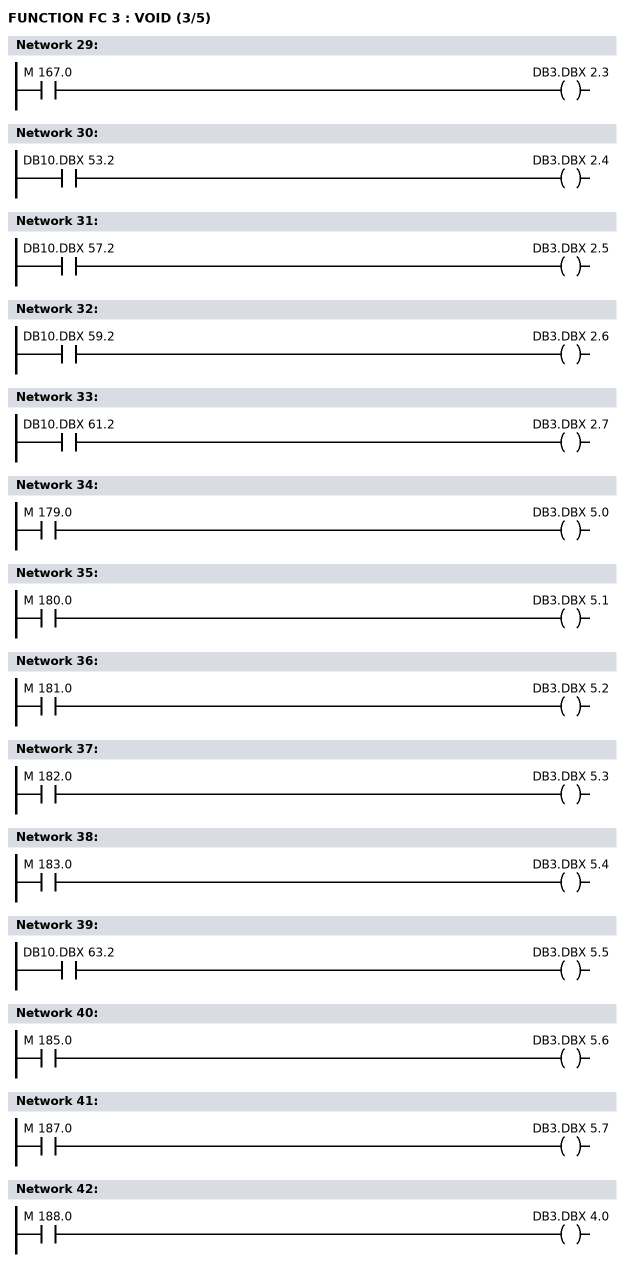

      A     M    167.0;
      =     DB3.DBX    2.3;
NETWORK
TITLE =

      A     DB10.DBX   53.2;
      =     DB3.DBX    2.4;
NETWORK
TITLE =

      A     DB10.DBX   57.2;
      =     DB3.DBX    2.5;
NETWORK
TITLE =

      A     DB10.DBX   59.2;
      =     DB3.DBX    2.6;
NETWORK
TITLE =

      A     DB10.DBX   61.2;
      =     DB3.DBX    2.7;
NETWORK
TITLE =

      A     M    179.0;
      =     DB3.DBX    5.0;
NETWORK
TITLE =

      A     M    180.0;
      =     DB3.DBX    5.1;
NETWORK
TITLE =

      A     M    181.0;
      =     DB3.DBX    5.2;
NETWORK
TITLE =

      A     M    182.0;
      =     DB3.DBX    5.3;
NETWORK
TITLE =

      A     M    183.0;
      =     DB3.DBX    5.4;
NETWORK
TITLE =

      A     DB10.DBX   63.2;
      =     DB3.DBX    5.5;
NETWORK
TITLE =

      A     M    185.0;
      =     DB3.DBX    5.6;
NETWORK
TITLE =

      A     M    187.0;
      =     DB3.DBX    5.7;
NETWORK
TITLE =

      A     M    188.0;
      =     DB3.DBX    4.0;
NETWORK
TITLE =
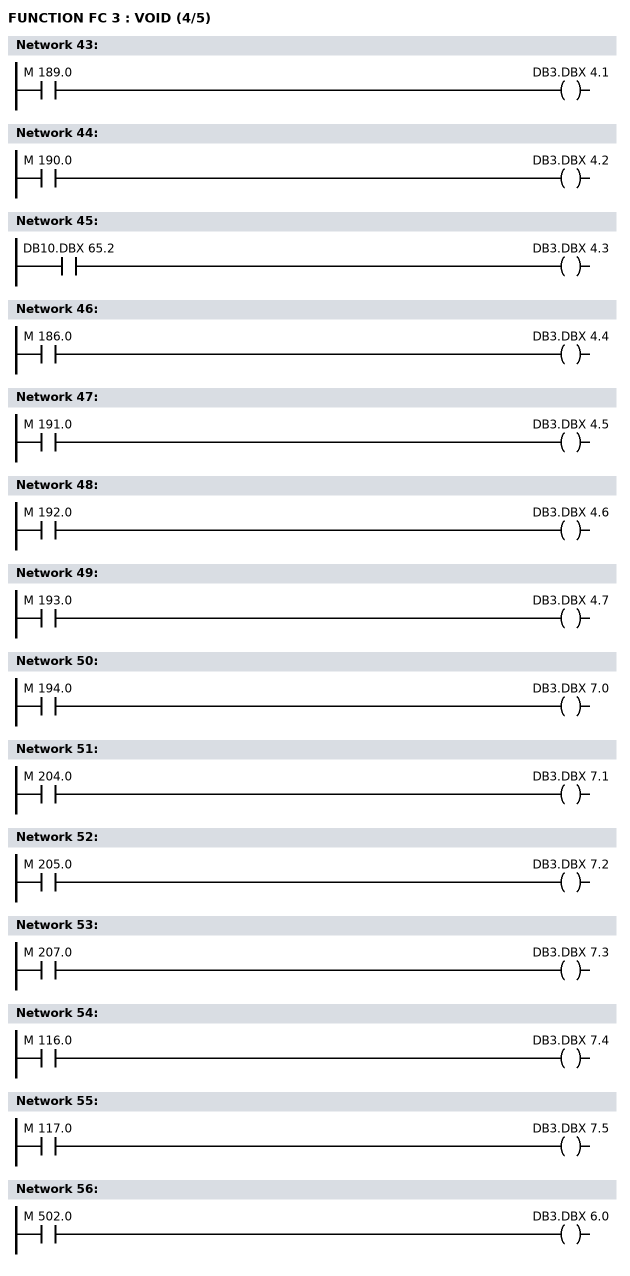

      A     M    189.0;
      =     DB3.DBX    4.1;
NETWORK
TITLE =

      A     M    190.0;
      =     DB3.DBX    4.2;
NETWORK
TITLE =

      A     DB10.DBX   65.2;
      =     DB3.DBX    4.3;
NETWORK
TITLE =

      A     M    186.0;
      =     DB3.DBX    4.4;
NETWORK
TITLE =

      A     M    191.0;
      =     DB3.DBX    4.5;
NETWORK
TITLE =

      A     M    192.0;
      =     DB3.DBX    4.6;
NETWORK
TITLE =

      A     M    193.0;
      =     DB3.DBX    4.7;
NETWORK
TITLE =

      A     M    194.0;
      =     DB3.DBX    7.0;
NETWORK
TITLE =

      A     M    204.0;
      =     DB3.DBX    7.1;
NETWORK
TITLE =

      A     M    205.0;
      =     DB3.DBX    7.2;
NETWORK
TITLE =

      A     M    207.0;
      =     DB3.DBX    7.3;
NETWORK
TITLE =

      A     M    116.0;
      =     DB3.DBX    7.4;
NETWORK
TITLE =

      A     M    117.0;
      =     DB3.DBX    7.5;
NETWORK
TITLE =

      A     M    502.0;
      =     DB3.DBX    6.0;
NETWORK
TITLE =
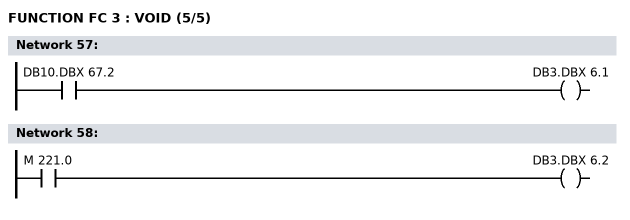

      A     DB10.DBX   67.2;
      =     DB3.DBX    6.1;
NETWORK
TITLE =

      A     M    221.0;
      =     DB3.DBX    6.2;
END_FUNCTION

FUNCTION FC 10 : VOID
TITLE =
AUTHOR : Xaadem <yalanci63@yahoo.com>
FAMILY : GENERAL
NAME : GENERAL
VERSION : 0.0


VAR_TEMP
  TEMP0 : BOOL ;
  TEMP1 : BOOL ;
  TEMP2 : BOOL ;
  TEMP3 : BOOL ;
END_VAR
BEGIN
NETWORK
TITLE =
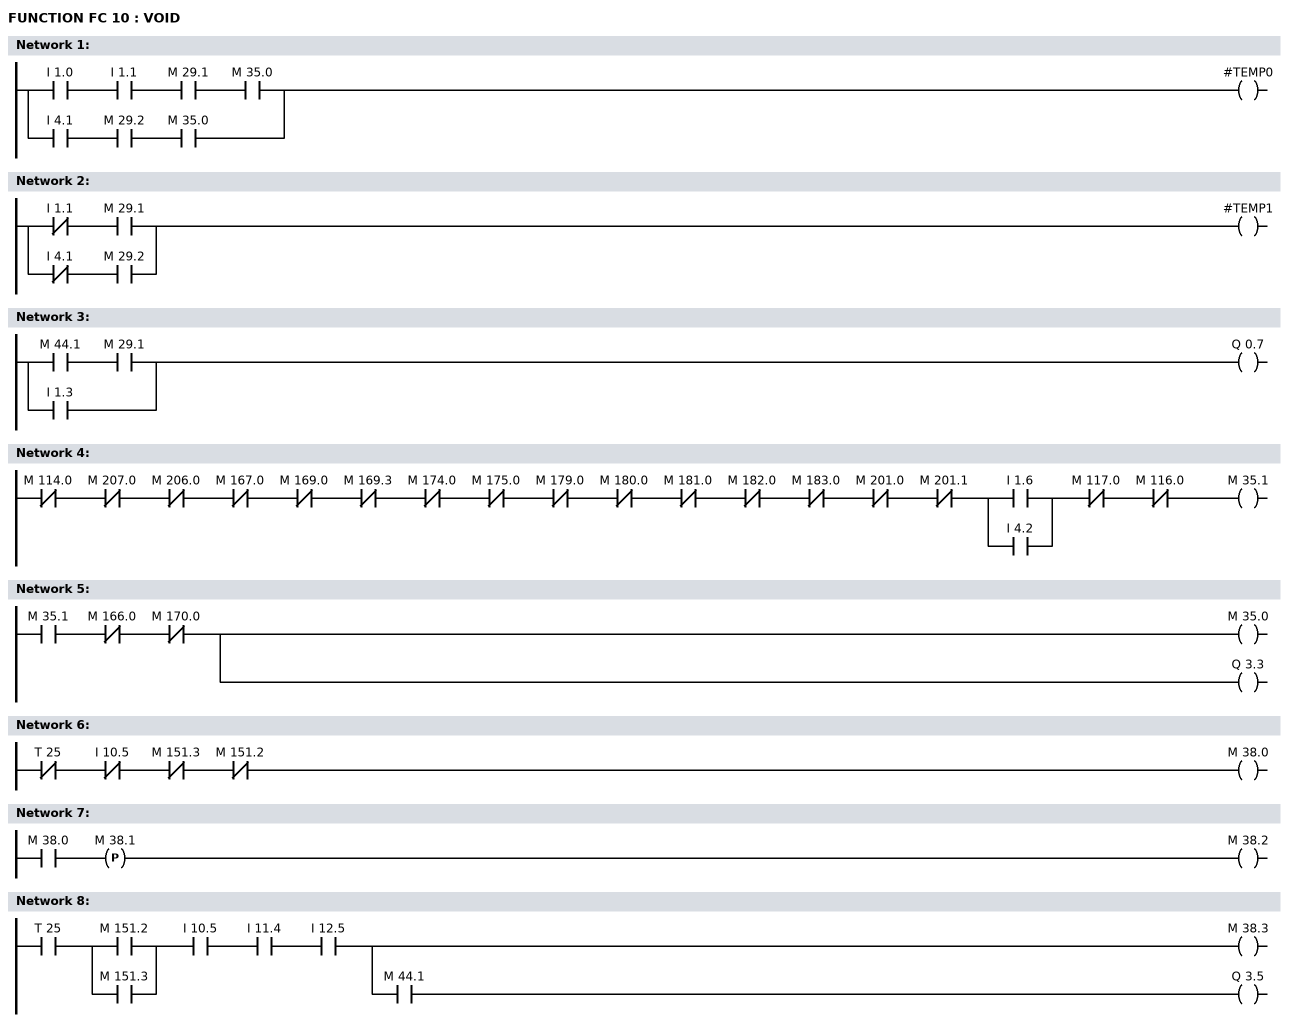

      A     I      1.0;
      A     I      1.1;
      A     M     29.1;
      A     M     35.0;
      O     ;
      A     I      4.1;
      A     M     29.2;
      A     M     35.0;
      =     #TEMP0;
NETWORK
TITLE =

      AN    I      1.1;
      A     M     29.1;
      O     ;
      AN    I      4.1;
      A     M     29.2;
      =     #TEMP1;
NETWORK
TITLE =

      A     M     44.1;
      A     M     29.1;
      O     I      1.3;
      =     Q      0.7;
NETWORK
TITLE =

      AN    M    114.0;
      AN    M    207.0;
      AN    M    206.0;
      AN    M    167.0;
      AN    M    169.0;
      AN    M    169.3;
      AN    M    174.0;
      AN    M    175.0;
      AN    M    179.0;
      AN    M    180.0;
      AN    M    181.0;
      AN    M    182.0;
      AN    M    183.0;
      AN    M    201.0;
      AN    M    201.1;
      A(    ;
      O     I      1.6;
      O     I      4.2;
      )     ;
      AN    M    117.0;
      AN    M    116.0;
      =     M     35.1;
NETWORK
TITLE =

      A     M     35.1;
      AN    M    166.0;
      AN    M    170.0;
      =     M     35.0;
      =     Q      3.3;
NETWORK
TITLE =

      AN    T     25;
      AN    I     10.5;
      AN    M    151.3;
      AN    M    151.2;
      =     M     38.0;
NETWORK
TITLE =

      A     M     38.0;
      FP    M     38.1;
      =     M     38.2;
NETWORK
TITLE =

      A     T     25;
      A(    ;
      O     M    151.2;
      O     M    151.3;
      )     ;
      A     I     10.5;
      A     I     11.4;
      A     I     12.5;
      =     L      1.0;
      A     L      1.0;
      BLD   102;
      =     M     38.3;
      A     L      1.0;
      A     M     44.1;
      =     Q      3.5;
NETWORK
TITLE =

      A(    ;
      A     M     35.0;
      A     #TEMP0;
      AN    #TEMP1;
      AN    M     38.3;
      FP    M     29.5;
      =     M     44.0;
      A     M     44.0;
      S     M     44.1;
      A(    ;
      O     M     20.7;
      ON    M     35.1;
      O     M     11.1;
      O     M     38.2;
      O     #TEMP1;
      O     M    114.0;
      )     ;
      R     M     44.1;
      A     M     44.1;
      )     ;
      A     M     38.3;
      O     ;
      AN    M     38.3;
      A     M     44.1;
      A     M     10.6;
      O     I      1.3;
      =     Q      3.1;
NETWORK
TITLE =
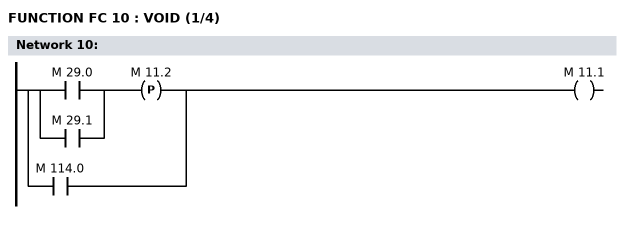

      A(    ;
      O     M     29.0;
      O     M     29.1;
      )     ;
      FP    M     11.2;
      O     M    114.0;
      =     M     11.1;
NETWORK
TITLE =
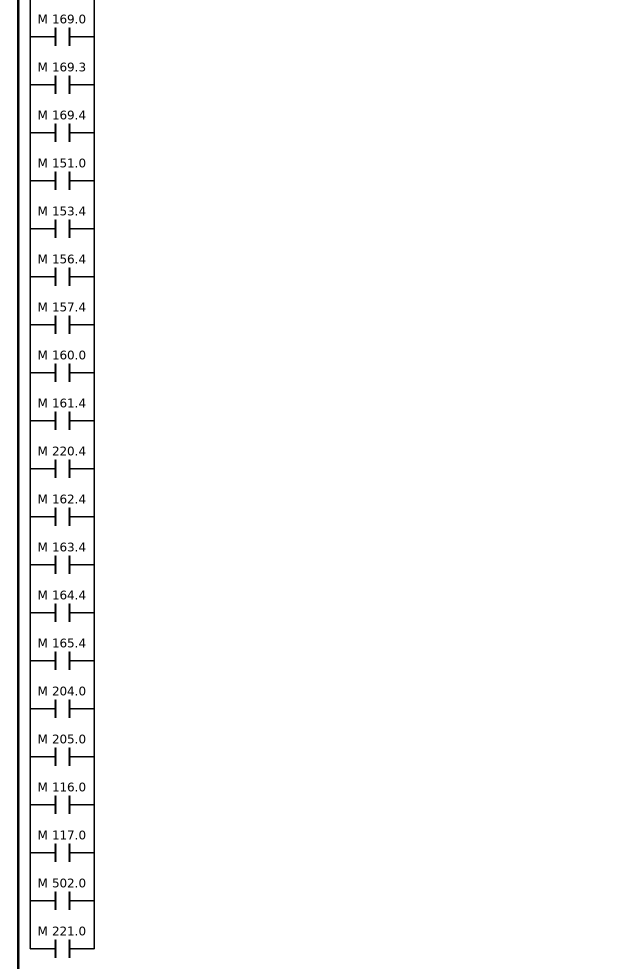

      O     M    155.0;
      O     M    155.1;
      O     M    158.0;
      O     M    166.0;
      O     M    167.0;
      O     M    170.0;
      O     M    174.0;
      O     M    175.0;
      O     M    179.0;
      O     M    180.0;
      O     M    181.0;
      O     M    182.0;
      O     M    183.0;
      O     M    185.0;
      O     M    186.0;
      O     M    187.0;
      O     M    188.0;
      O     M    189.0;
      O     M    190.0;
      O     M    191.0;
      O     M    192.0;
      O     M    193.0;
      O     M    194.0;
      O     M    195.0;
      O     M    196.0;
      O     M    198.0;
      O     M    197.0;
      O     M    199.0;
      O     M    169.0;
      O     M    169.3;
      O     M    169.4;
      O     M    151.0;
      O     M    153.4;
      O     M    156.4;
      O     M    157.4;
      O     M    160.0;
      O     M    161.4;
      O     M    220.4;
      O     M    162.4;
      O     M    163.4;
      O     M    164.4;
      O     M    165.4;
      O     M    204.0;
      O     M    205.0;
      O     M    116.0;
      O     M    117.0;
      O     M    502.0;
      O     M    221.0;
      =     M     24.0;
NETWORK
TITLE =
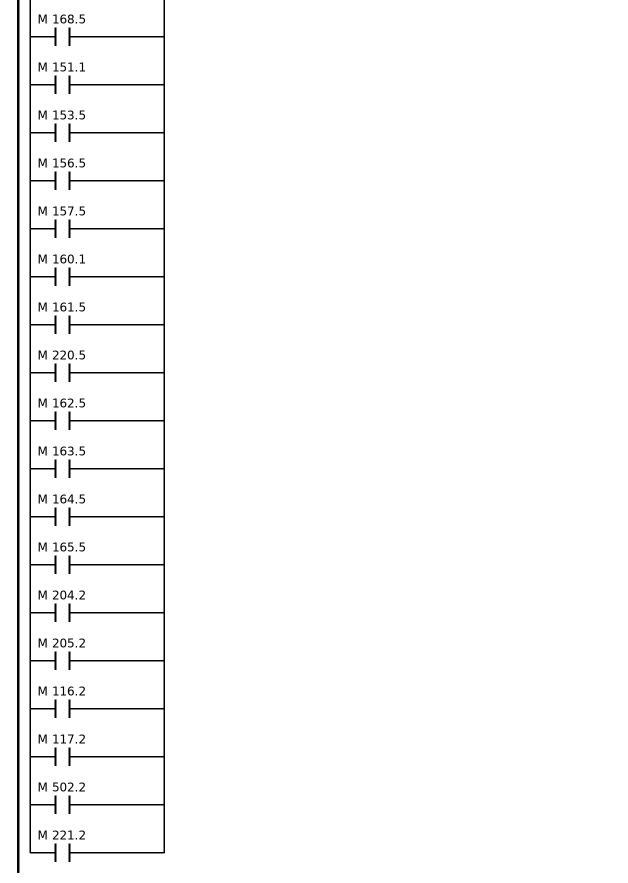

      O     M    155.2;
      O(    ;
      A     M    155.1;
      FP    M    155.3;
      )     ;
      O     M    158.2;
      O     M    166.2;
      O     M    167.2;
      O     M    170.2;
      O     M    174.2;
      O     M    175.2;
      O     M    179.2;
      O     M    180.2;
      O     M    181.2;
      O     M    182.2;
      O     M    183.2;
      O     M    185.2;
      O     M    186.2;
      O     M    187.2;
      O     M    188.2;
      O     M    189.2;
      O     M    190.2;
      O     M    191.2;
      O     M    192.2;
      O     M    193.2;
      O     M    194.2;
      O     M    195.2;
      O     M    196.2;
      O     M    198.2;
      O     M    197.2;
      O     M    199.2;
      O     M    168.5;
      O     M    151.1;
      O     M    153.5;
      O     M    156.5;
      O     M    157.5;
      O     M    160.1;
      O     M    161.5;
      O     M    220.5;
      O     M    162.5;
      O     M    163.5;
      O     M    164.5;
      O     M    165.5;
      O     M    204.2;
      O     M    205.2;
      O     M    116.2;
      O     M    117.2;
      O     M    502.2;
      O     M    221.2;
      =     M     22.0;
NETWORK
TITLE =
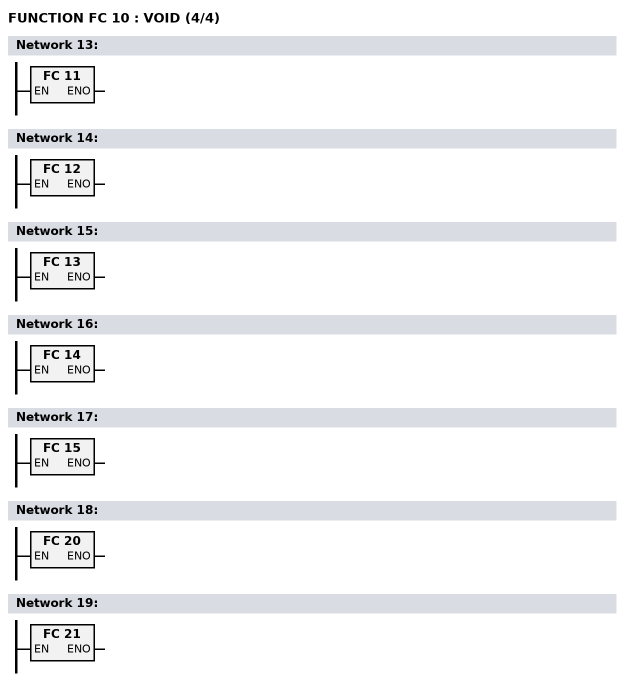

      CALL FC    11 ;
      NOP   0;
NETWORK
TITLE =

      CALL FC    12 ;
      NOP   0;
NETWORK
TITLE =

      CALL FC    13 ;
      NOP   0;
NETWORK
TITLE =

      CALL FC    14 ;
      NOP   0;
NETWORK
TITLE =

      CALL FC    15 ;
      NOP   0;
NETWORK
TITLE =

      CALL FC    20 ;
      NOP   0;
NETWORK
TITLE =

      CALL FC    21 ;
      NOP   0;
END_FUNCTION

FUNCTION_BLOCK FB 42
TITLE =
AUTHOR : Xaadem <yalanci63@yahoo.com>
NAME : PID
VERSION : 0.1


VAR_INPUT
  IN0 : BOOL ;
  IN1 : BOOL ;
  IN2 : BOOL ;
  IN3 : BOOL ;
  IN4 : BOOL ;
  IN5 : BOOL ;
  IN6 : BOOL ;
  IN7 : TIME  := T#1S;
  IN8 : REAL ;
  IN9 : REAL ;
  IN10 : WORD ;
  IN11 : REAL  := 2.000000e+000;
  IN12 : TIME  := T#20S;
  IN13 : REAL  := 1.000000e+000;
  IN14 : REAL  := 1.000000e+000;
  IN15 : REAL ;
  IN16 : TIME  := T#3S;
  IN17 : TIME  := T#3S;
  IN18 : TIME  := T#30S;
  IN19 : REAL ;
END_VAR
VAR_OUTPUT
  OUT20 : BOOL ;
  OUT21 : BOOL ;
  OUT22 : REAL ;
  OUT23 : REAL ;
END_VAR
VAR
  STAT24 : BOOL ;
  STAT25 : REAL ;
  STAT26 : REAL ;
  STAT27 : REAL ;
  STAT28 : REAL ;
  STAT29 : INT ;
  STAT30 : TIME ;
  STAT31 : TIME ;
END_VAR
VAR_TEMP
  TEMP32 : REAL ;
  TEMP33 : REAL ;
  TEMP41 : REAL ;
  TEMP34 : REAL ;
  TEMP35 : REAL ;
  TEMP36 : REAL ;
  TEMP37 : REAL ;
  TEMP38 : REAL ;
  TEMP39 : INT ;
  TEMP40 : REAL ;
  TEMP42 : REAL ;
  TEMP43 : REAL ;
  TEMP44 : REAL ;
END_VAR
BEGIN
NETWORK
TITLE =

      SET   ;
      SAVE  ;
      =     L     50.1;
      A     #IN0;
      JCN   M001;
      L     #STAT25;
      T     #STAT26;
      CLR   ;
      =     #OUT20;
      =     #OUT21;
      L     0.000000e+000;
      T     #OUT22;
      T     #OUT23;
      =     #STAT24;
      T     #STAT25;
      T     #STAT26;
      T     #STAT27;
      T     #STAT28;
      L     0;
      T     #STAT29;
      L     T#0MS;
      T     #STAT30;
      T     #STAT31;
      JU    M002;
M001: L     #IN10;
      ITD   ;
      DTR   ;
      L     3.616898e-003;
      *R    ;
      T     #TEMP34;
      L     #IN14;
      *R    ;
      L     #IN15;
      +R    ;
      T     #TEMP34;
      CLR   ;
      A     #IN6;
      NOT   ;
      JCN   M003;
      L     #IN9;
      T     #TEMP34;
M003: L     #TEMP34;
      T     #OUT22;
      L     #IN8;
      TAK   ;
      -R    ;
      T     #TEMP35;
      L     #IN13;
      NEGR  ;
      <R    ;
      JCN   M004;
      TAK   ;
      L     #IN13;
      +R    ;
      T     #OUT23;
      JU    M005;
M004: L     #TEMP35;
      L     #IN13;
      >R    ;
      JCN   M006;
      -R    ;
      T     #OUT23;
      JU    M005;
M006: L     0.000000e+000;
      T     #OUT23;
M005: L     #OUT23;
      L     #IN11;
      *R    ;
      T     #TEMP35;
      L     #IN7;
      DTR   ;
      L     1.000000e+003;
      /R    ;
      T     #TEMP33;
      L     #IN12;
      DTR   ;
      L     1.000000e+003;
      /R    ;
      T     #TEMP36;
      L     #TEMP33;
      L     5.000000e-001;
      *R    ;
      L     #TEMP36;
      TAK   ;
      <R    ;
      JCN   M007;
      L     #TEMP33;
      L     5.000000e-001;
      *R    ;
      T     #TEMP36;
M007: L     #IN18;
      DTR   ;
      L     1.000000e+003;
      /R    ;
      T     #TEMP40;
      L     1.000000e-002;
      L     #TEMP35;
      *R    ;
      L     #TEMP40;
      *R    ;
      ABS   ;
      L     #TEMP36;
      TAK   ;
      -R    ;
      T     #TEMP32;
      L     1.000000e-001;
      L     #TEMP36;
      *R    ;
      L     #TEMP32;
      TAK   ;
      <R    ;
      JCN   M008;
      L     1.000000e-001;
      L     #TEMP36;
      *R    ;
      T     #TEMP36;
      JU    M009;
M008: L     #TEMP32;
      T     #TEMP36;
M009: CLR   ;
      A     #IN3;
      JCN   M00a;
      L     0.000000e+000;
      T     #STAT27;
      JU    M00b;
M00a: L     #STAT29;
      L     0;
      <>I   ;
      JCN   M00c;
      TAK   ;
      ITD   ;
      DTR   ;
      L     #TEMP33;
      *R    ;
      L     #TEMP40;
      /R    ;
      T     #TEMP42;
      JU    M00d;
M00c: L     #TEMP35;
      L     0.000000e+000;
      >R    ;
      A     #IN1;
      =     L     50.2;
      <R    ;
      A     #IN2;
      O     L     50.2;
      L     #IN12;
      L     T#0MS;
      =     L     50.2;
      ==D   ;
      O     L     50.2;
      JCN   M00e;
      L     0.000000e+000;
      T     #TEMP42;
      JU    M00d;
M00e: L     #TEMP35;
      NEGR  ;
      L     #TEMP33;
      *R    ;
      L     #TEMP36;
      /R    ;
      T     #TEMP42;
M00d: L     #STAT27;
      L     #TEMP42;
      +R    ;
      T     #STAT27;
      L     #IN12;
      L     T#0MS;
      ==D   ;
      JCN   M00b;
      L     #STAT27;
      L     1.000000e+002;
      >R    ;
      JCN   M00f;
      T     #STAT27;
      JU    M00b;
M00f: L     #STAT27;
      L     0.000000e+000;
      <R    ;
      JCN   M00b;
      T     #STAT27;
M00b: L     #TEMP35;
      L     #STAT27;
      -R    ;
      L     #IN19;
      +R    ;
      T     #TEMP43;
      L     #TEMP35;
      T     #TEMP37;
      L     #STAT27;
      T     #TEMP38;
      L     5.500000e+001;
      L     #TEMP40;
      /R    ;
      L     #TEMP33;
      *R    ;
      T     #TEMP41;
      L     #IN16;
      L     #IN7;
      >D    ;
      JCN   M010;
      TAK   ;
      DTR   ;
      L     1.000000e+003;
      /R    ;
      T     #TEMP32;
      JU    M011;
M010: L     #TEMP33;
      T     #TEMP32;
M011: L     1.000000e+002;
      L     #TEMP32;
      *R    ;
      L     #TEMP40;
      /R    ;
      T     #TEMP32;
      CLR   ;
      A     #IN1;
      O     #IN2;
      NOT   ;
      JCN   M012;
      A     #OUT20;
      O     #OUT21;
      NOT   ;
      JCN   M013;
      L     #IN12;
      L     T#0MS;
      <>D   ;
      JCN   M014;
      L     #TEMP37;
      ABS   ;
      T     #TEMP37;
      L     #TEMP38;
      ABS   ;
      T     #TEMP38;
      <R    ;
      JCN   M015;
      TAK   ;
      T     #STAT28;
      JU    M016;
M015: L     #TEMP38;
      T     #STAT28;
      JU    M016;
M014: L     #TEMP34;
      L     0.000000e+000;
      ==R   ;
      JCN   M017;
      L     #TEMP32;
      T     #STAT28;
      JU    M016;
M017: L     #TEMP35;
      ABS   ;
      L     5.000000e-001;
      *R    ;
      T     #STAT28;
M016: L     #STAT28;
      L     1.000000e+001;
      >R    ;
      JCN   M018;
      T     #STAT28;
M018: L     #STAT28;
      L     #TEMP32;
      <R    ;
      JCN   M019;
      T     #STAT28;
M019: JU    M013;
M012: L     #TEMP32;
      T     #STAT28;
M013: L     #STAT29;
      L     100;
      ==I   ;
      L     #TEMP43;
      L     #TEMP41;
      =     L     50.2;
      >R    ;
      A     L     50.2;
      TAK   ;
      L     #STAT28;
      =     L     50.2;
      >=R   ;
      O     L     50.2;
      JCN   M01a;
      L     100;
      T     #TEMP39;
      JU    M01b;
M01a: L     #STAT29;
      L     -100;
      ==I   ;
      L     #TEMP41;
      NEGR  ;
      L     #TEMP43;
      TAK   ;
      =     L     50.2;
      <R    ;
      A     L     50.2;
      L     #STAT28;
      NEGR  ;
      L     #TEMP43;
      TAK   ;
      =     L     50.2;
      <=R   ;
      O     L     50.2;
      JCN   M01c;
      L     -100;
      T     #TEMP39;
      JU    M01b;
M01c: L     0;
      T     #TEMP39;
M01b: CLR   ;
      A     #IN3;
      JCN   M01d;
      A     #IN4;
      X     #IN5;
      JCN   M01e;
      A     #IN4;
      JCN   M01f;
      L     100;
      T     #TEMP39;
      JU    M01d;
M01f: L     -100;
      T     #TEMP39;
      JU    M01d;
M01e: L     0;
      T     #TEMP39;
M01d: L     #TEMP39;
      L     100;
      ==I   ;
      A     #IN1;
      TAK   ;
      L     -100;
      =     L     50.2;
      ==I   ;
      A     #IN2;
      O     L     50.2;
      JCN   M020;
      L     0;
      T     #TEMP39;
M020: L     #STAT29;
      L     -100;
      ==I   ;
      L     #TEMP39;
      L     100;
      =     L     50.2;
      ==I   ;
      A     L     50.2;
      L     #STAT29;
      TAK   ;
      =     L     50.2;
      ==I   ;
      L     #TEMP39;
      L     -100;
      =     L     50.3;
      ==I   ;
      A     L     50.3;
      O     L     50.2;
      JCN   M021;
      L     0;
      T     #TEMP39;
M021: L     #STAT29;
      L     #TEMP39;
      <>I   ;
      JCN   M022;
      L     0;
      ==I   ;
      JCN   M023;
      L     #STAT30;
      L     T#0MS;
      <=D   ;
      JCN   M022;
      L     0;
      T     #STAT29;
      L     #IN17;
      T     #STAT31;
      JU    M022;
M023: L     #STAT31;
      L     T#0MS;
      <=D   ;
      JCN   M022;
      L     #TEMP39;
      T     #STAT29;
      L     #IN16;
      T     #STAT30;
M022: L     #STAT30;
      L     T#0MS;
      >D    ;
      JCN   M024;
      TAK   ;
      L     #IN7;
      -D    ;
      T     #STAT30;
      JU    M025;
M024: L     T#0MS;
      T     #STAT30;
M025: L     #STAT31;
      L     T#0MS;
      >D    ;
      JCN   M026;
      TAK   ;
      L     #IN7;
      -D    ;
      T     #STAT31;
      JU    M027;
M026: L     T#0MS;
      T     #STAT31;
M027: L     #STAT29;
      L     100;
      ==I   ;
      A     #IN1;
      TAK   ;
      L     -100;
      =     L     50.2;
      ==I   ;
      A     #IN2;
      O     L     50.2;
      JCN   M028;
      L     0;
      T     #STAT29;
      L     T#0MS;
      T     #STAT30;
M028: CLR   ;
      A     #STAT24;
      NOT   ;
      JCN   M029;
      L     #STAT25;
      T     #TEMP44;
      JU    M02a;
M029: L     #STAT29;
      ITD   ;
      DTR   ;
      L     #TEMP33;
      *R    ;
      L     #TEMP40;
      /R    ;
      L     #STAT26;
      +R    ;
      T     #TEMP44;
      L     1.000000e+002;
      >=R   ;
      JCN   M02b;
      T     #TEMP44;
      JU    M02a;
M02b: L     #TEMP44;
      L     0.000000e+000;
      <=R   ;
      JCN   M02a;
      T     #TEMP44;
M02a: L     #TEMP44;
      T     #STAT26;
      L     #STAT29;
      L     0;
      ==I   ;
      JCN   M02c;
      CLR   ;
      =     #OUT20;
      =     #OUT21;
      JU    M002;
M02c: L     #STAT29;
      L     100;
      ==I   ;
      JCN   M02d;
      SET   ;
      =     #OUT20;
      CLR   ;
      =     #OUT21;
      JU    M002;
M02d: CLR   ;
      =     #OUT20;
      SET   ;
      =     #OUT21;
M002: CLR   ;
      A     L     50.1;
      SAVE  ;
      BE    ;


END_FUNCTION_BLOCK

DATA_BLOCK DB 18
TITLE =
AUTHOR : Xaadem <yalanci63@yahoo.com>
FAMILY : CONTROLL
NAME : 'DB'
VERSION : 0.0

 FB 42
BEGIN
   IN0 := FALSE;
   IN1 := FALSE;
   IN2 := FALSE;
   IN3 := FALSE;
   IN4 := FALSE;
   IN5 := FALSE;
   IN6 := FALSE;
   IN7 := T#1S;
   IN8 := 0.000000e+000;
   IN9 := -4.200000e+001;
   IN10 := W#16#0;
   IN11 := 5.000000e-001;
   IN12 := T#10S;
   IN13 := 5.000000e+001;
   IN14 := 1.000000e+000;
   IN15 := 0.000000e+000;
   IN16 := T#500MS;
   IN17 := T#1S;
   IN18 := T#30S;
   IN19 := 0.000000e+000;
   OUT20 := FALSE;
   OUT21 := FALSE;
   OUT22 := -4.200000e+001;
   OUT23 := 0.000000e+000;
   STAT24 := FALSE;
   STAT25 := 0.000000e+000;
   STAT26 := 0.000000e+000;
   STAT27 := 7.902575e-001;
   STAT28 := 3.333333e+000;
   STAT29 := 0;
   STAT30 := T#0MS;
   STAT31 := T#0MS;
END_DATA_BLOCK

FUNCTION FC 191 : VOID
TITLE =
AUTHOR : Xaadem <yalanci63@yahoo.com>
FAMILY : ZE
NAME : S
VERSION : 0.0


VAR_INPUT
  IN0 : BOOL ;
  IN1 : BOOL ;
END_VAR
VAR_IN_OUT
  IO2 : INT ;
  IO3 : INT ;
  IO4 : INT ;
  IO5 : INT ;
  IO6 : INT ;
  IO7 : WORD ;
END_VAR
VAR_TEMP
  TEMP8 : BOOL ;
  TEMP9 : BOOL ;
  TEMP10 : BOOL ;
  TEMP11 : BOOL ;
  TEMP12 : BOOL ;
END_VAR
BEGIN
NETWORK
TITLE =
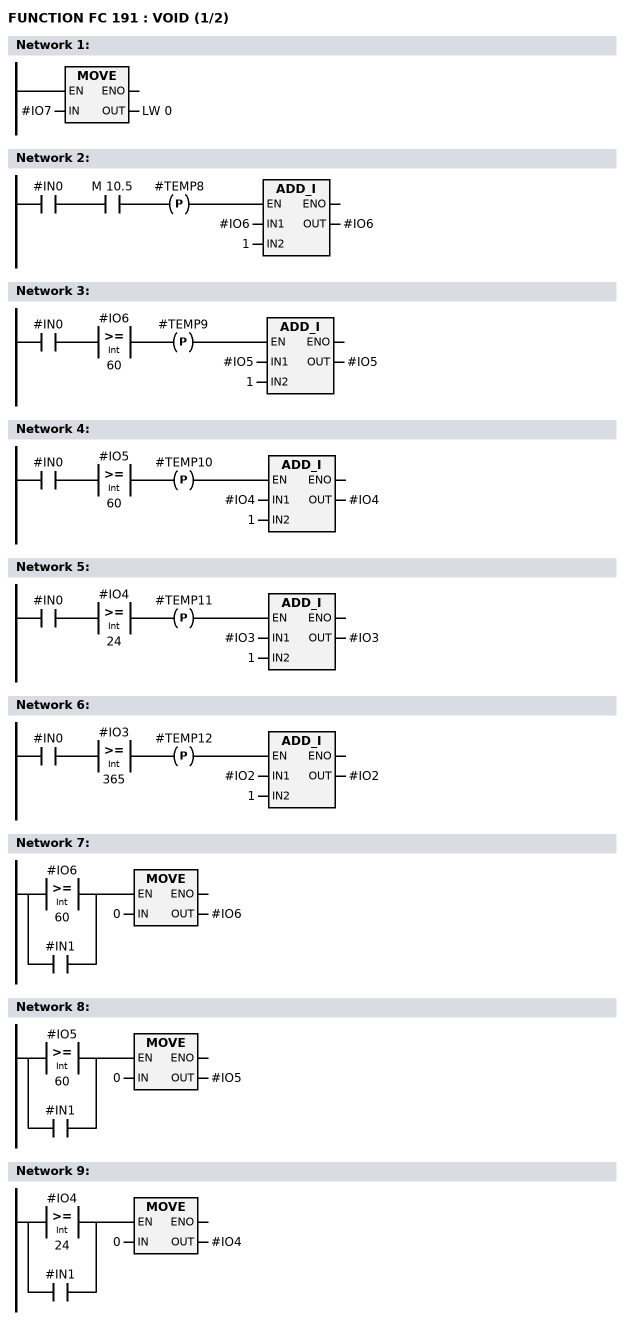

      L     #IO7;
      T     LW     0;
      NOP   0;
NETWORK
TITLE =

      A     #IN0;
      A     M     10.5;
      FP    #TEMP8;
      JNB   M001;
      L     #IO6;
      L     1;
      +I    ;
      T     #IO6;
M001: NOP   0;
NETWORK
TITLE =

      A     #IN0;
      A(    ;
      L     #IO6;
      L     60;
      >=I   ;
      )     ;
      FP    #TEMP9;
      JNB   M002;
      L     #IO5;
      L     1;
      +I    ;
      T     #IO5;
M002: NOP   0;
NETWORK
TITLE =

      A     #IN0;
      A(    ;
      L     #IO5;
      L     60;
      >=I   ;
      )     ;
      FP    #TEMP10;
      JNB   M003;
      L     #IO4;
      L     1;
      +I    ;
      T     #IO4;
M003: NOP   0;
NETWORK
TITLE =

      A     #IN0;
      A(    ;
      L     #IO4;
      L     24;
      >=I   ;
      )     ;
      FP    #TEMP11;
      JNB   M004;
      L     #IO3;
      L     1;
      +I    ;
      T     #IO3;
M004: NOP   0;
NETWORK
TITLE =

      A     #IN0;
      A(    ;
      L     #IO3;
      L     365;
      >=I   ;
      )     ;
      FP    #TEMP12;
      JNB   M005;
      L     #IO2;
      L     1;
      +I    ;
      T     #IO2;
M005: NOP   0;
NETWORK
TITLE =

      A(    ;
      O(    ;
      L     #IO6;
      L     60;
      >=I   ;
      )     ;
      O     #IN1;
      )     ;
      JNB   M006;
      L     0;
      T     #IO6;
M006: NOP   0;
NETWORK
TITLE =

      A(    ;
      O(    ;
      L     #IO5;
      L     60;
      >=I   ;
      )     ;
      O     #IN1;
      )     ;
      JNB   M007;
      L     0;
      T     #IO5;
M007: NOP   0;
NETWORK
TITLE =

      A(    ;
      O(    ;
      L     #IO4;
      L     24;
      >=I   ;
      )     ;
      O     #IN1;
      )     ;
      JNB   M008;
      L     0;
      T     #IO4;
M008: NOP   0;
NETWORK
TITLE =
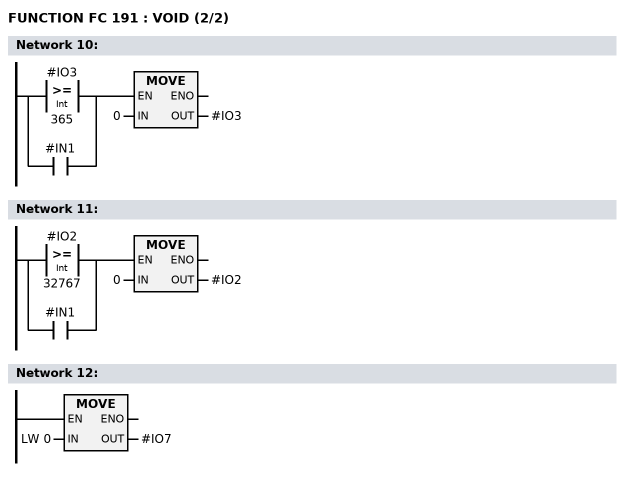

      A(    ;
      O(    ;
      L     #IO3;
      L     365;
      >=I   ;
      )     ;
      O     #IN1;
      )     ;
      JNB   M009;
      L     0;
      T     #IO3;
M009: NOP   0;
NETWORK
TITLE =

      A(    ;
      O(    ;
      L     #IO2;
      L     32767;
      >=I   ;
      )     ;
      O     #IN1;
      )     ;
      JNB   M00a;
      L     0;
      T     #IO2;
M00a: NOP   0;
NETWORK
TITLE =

      L     LW     0;
      T     #IO7;
      NOP   0;
END_FUNCTION

FUNCTION FC 1 : VOID
TITLE =
AUTHOR : Xaadem <yalanci63@yahoo.com>
FAMILY : GENERAL
NAME : GENERAL
VERSION : 0.0

BEGIN
NETWORK
TITLE =
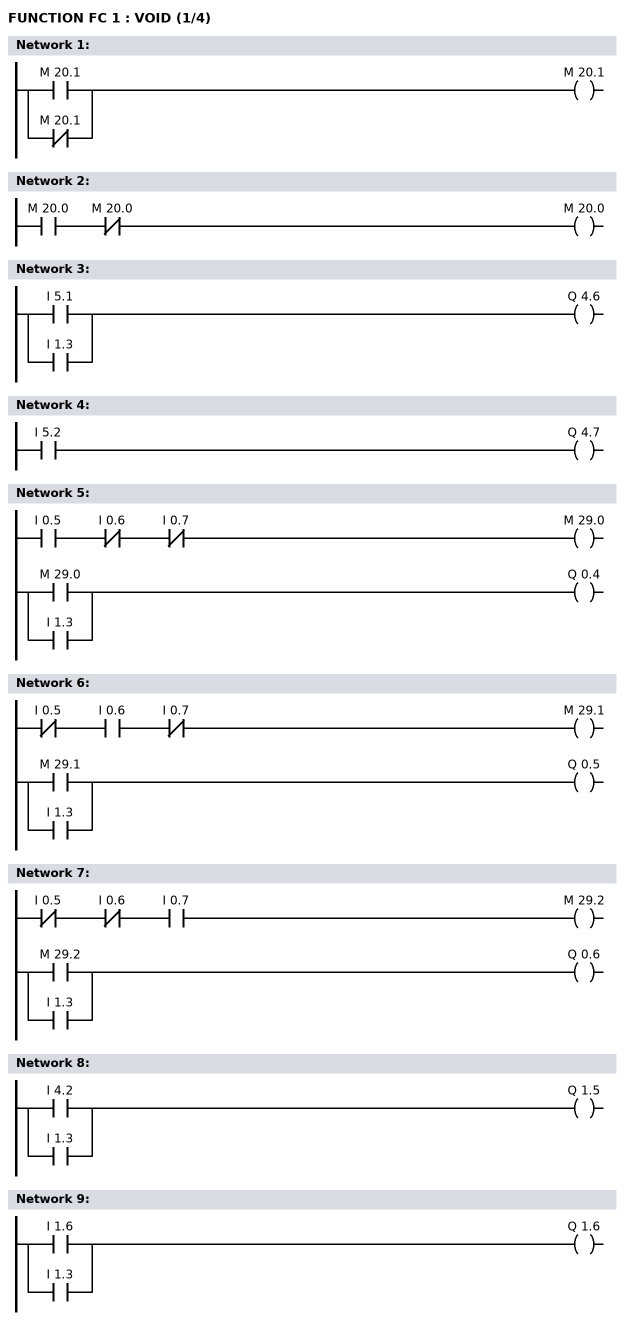

      O     M     20.1;
      ON    M     20.1;
      =     M     20.1;
NETWORK
TITLE =

      A     M     20.0;
      AN    M     20.0;
      =     M     20.0;
NETWORK
TITLE =

      O     I      5.1;
      O     I      1.3;
      =     Q      4.6;
NETWORK
TITLE =

      A     I      5.2;
      =     Q      4.7;
NETWORK
TITLE =

      A     I      0.5;
      AN    I      0.6;
      AN    I      0.7;
      =     M     29.0;
      A     M     29.0;
      O     I      1.3;
      =     Q      0.4;
NETWORK
TITLE =

      AN    I      0.5;
      A     I      0.6;
      AN    I      0.7;
      =     M     29.1;
      A     M     29.1;
      O     I      1.3;
      =     Q      0.5;
NETWORK
TITLE =

      AN    I      0.5;
      AN    I      0.6;
      A     I      0.7;
      =     M     29.2;
      A     M     29.2;
      O     I      1.3;
      =     Q      0.6;
NETWORK
TITLE =

      O     I      4.2;
      O     I      1.3;
      =     Q      1.5;
NETWORK
TITLE =

      O     I      1.6;
      O     I      1.3;
      =     Q      1.6;
NETWORK
TITLE =
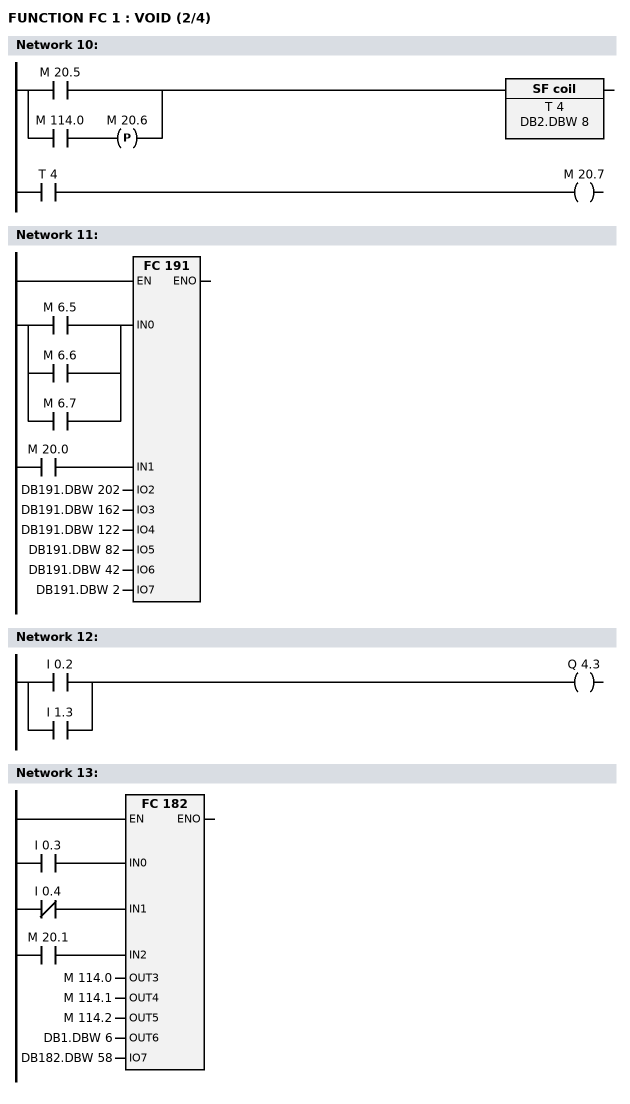

      A(    ;
      O     M     20.5;
      O(    ;
      A     M    114.0;
      FP    M     20.6;
      )     ;
      )     ;
      L     DB2.DBW    8;
      SF    T      4;
      NOP   0;
      NOP   0;
      NOP   0;
      A     T      4;
      =     M     20.7;
NETWORK
TITLE =

      A(    ;
      O     M      6.5;
      O     M      6.6;
      O     M      6.7;
      )     ;
      =     L      0.0;
      BLD   103;
      A     M     20.0;
      =     L      0.1;
      BLD   103;
      CALL FC   191 (
           IN0                      := L      0.0,
           IN1                      := L      0.1,
           IO2                      := DB191.DBW  202,
           IO3                      := DB191.DBW  162,
           IO4                      := DB191.DBW  122,
           IO5                      := DB191.DBW   82,
           IO6                      := DB191.DBW   42,
           IO7                      := DB191.DBW    2);
      NOP   0;
NETWORK
TITLE =

      O     I      0.2;
      O     I      1.3;
      =     Q      4.3;
NETWORK
TITLE =

      A     I      0.3;
      =     L      0.0;
      BLD   103;
      AN    I      0.4;
      =     L      0.1;
      BLD   103;
      A     M     20.1;
      =     L      0.2;
      BLD   103;
      CALL FC   182 (
           IN0                      := L      0.0,
           IN1                      := L      0.1,
           IN2                      := L      0.2,
           OUT3                     := M    114.0,
           OUT4                     := M    114.1,
           OUT5                     := M    114.2,
           OUT6                     := DB1.DBW    6,
           IO7                      := DB182.DBW   58);
      NOP   0;
NETWORK
TITLE =
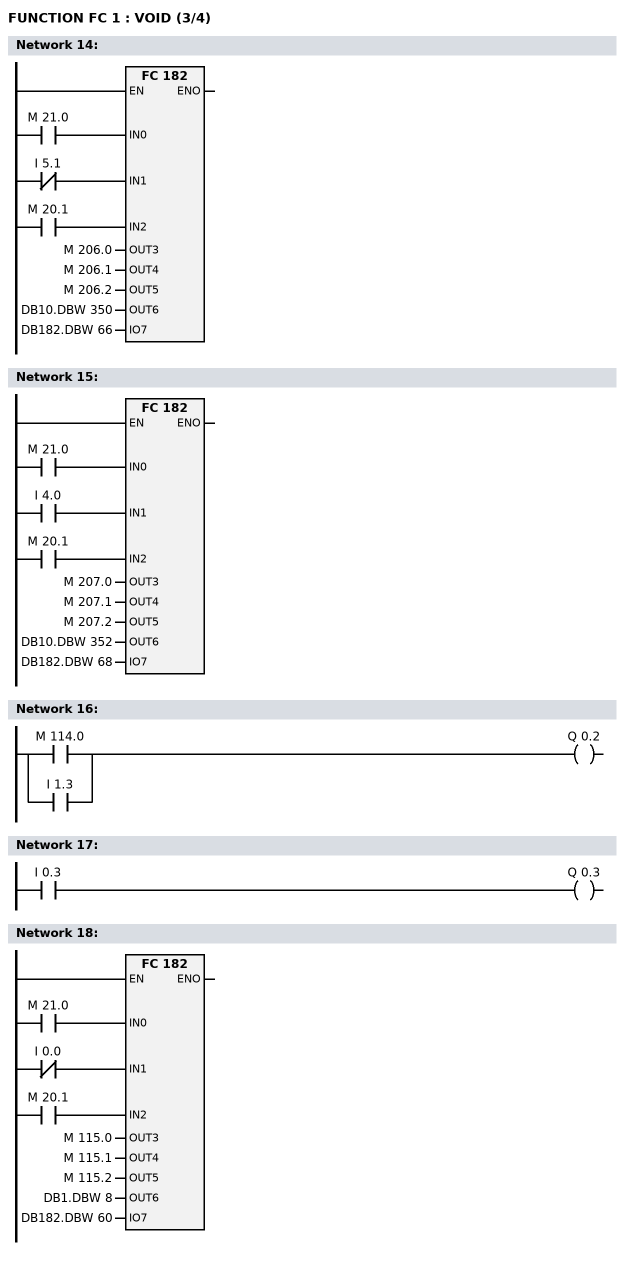

      A     M     21.0;
      =     L      0.0;
      BLD   103;
      AN    I      5.1;
      =     L      0.1;
      BLD   103;
      A     M     20.1;
      =     L      0.2;
      BLD   103;
      CALL FC   182 (
           IN0                      := L      0.0,
           IN1                      := L      0.1,
           IN2                      := L      0.2,
           OUT3                     := M    206.0,
           OUT4                     := M    206.1,
           OUT5                     := M    206.2,
           OUT6                     := DB10.DBW  350,
           IO7                      := DB182.DBW   66);
      NOP   0;
NETWORK
TITLE =

      A     M     21.0;
      =     L      0.0;
      BLD   103;
      A     I      4.0;
      =     L      0.1;
      BLD   103;
      A     M     20.1;
      =     L      0.2;
      BLD   103;
      CALL FC   182 (
           IN0                      := L      0.0,
           IN1                      := L      0.1,
           IN2                      := L      0.2,
           OUT3                     := M    207.0,
           OUT4                     := M    207.1,
           OUT5                     := M    207.2,
           OUT6                     := DB10.DBW  352,
           IO7                      := DB182.DBW   68);
      NOP   0;
NETWORK
TITLE =

      O     M    114.0;
      O     I      1.3;
      =     Q      0.2;
NETWORK
TITLE =

      A     I      0.3;
      =     Q      0.3;
NETWORK
TITLE =

      A     M     21.0;
      =     L      0.0;
      BLD   103;
      AN    I      0.0;
      =     L      0.1;
      BLD   103;
      A     M     20.1;
      =     L      0.2;
      BLD   103;
      CALL FC   182 (
           IN0                      := L      0.0,
           IN1                      := L      0.1,
           IN2                      := L      0.2,
           OUT3                     := M    115.0,
           OUT4                     := M    115.1,
           OUT5                     := M    115.2,
           OUT6                     := DB1.DBW    8,
           IO7                      := DB182.DBW   60);
      NOP   0;
NETWORK
TITLE =
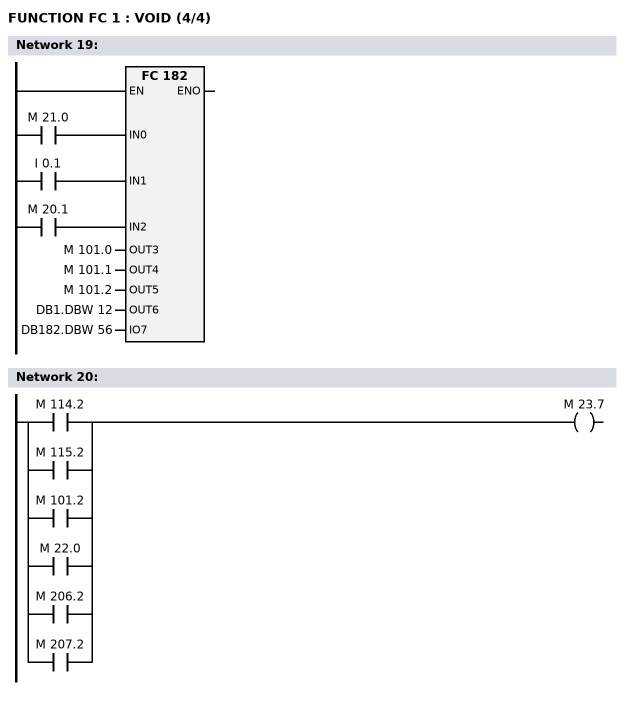

      A     M     21.0;
      =     L      0.0;
      BLD   103;
      A     I      0.1;
      =     L      0.1;
      BLD   103;
      A     M     20.1;
      =     L      0.2;
      BLD   103;
      CALL FC   182 (
           IN0                      := L      0.0,
           IN1                      := L      0.1,
           IN2                      := L      0.2,
           OUT3                     := M    101.0,
           OUT4                     := M    101.1,
           OUT5                     := M    101.2,
           OUT6                     := DB1.DBW   12,
           IO7                      := DB182.DBW   56);
      NOP   0;
NETWORK
TITLE =

      O     M    114.2;
      O     M    115.2;
      O     M    101.2;
      O     M     22.0;
      O     M    206.2;
      O     M    207.2;
      =     M     23.7;
NETWORK
TITLE =

      O     M    114.0;
      O     M    115.0;
      O     M    101.0;
      O     M     24.0;
      O     M    206.0;
      O     M    207.0;
      =     L      0.0;
      O     L      0.0;
      O     I      1.3;
      =     Q      1.0;
      A     L      0.0;
      BLD   102;
      =     Q      0.1;
      A     L      0.0;
      BLD   102;
      =     Q      3.4;
NETWORK
TITLE =
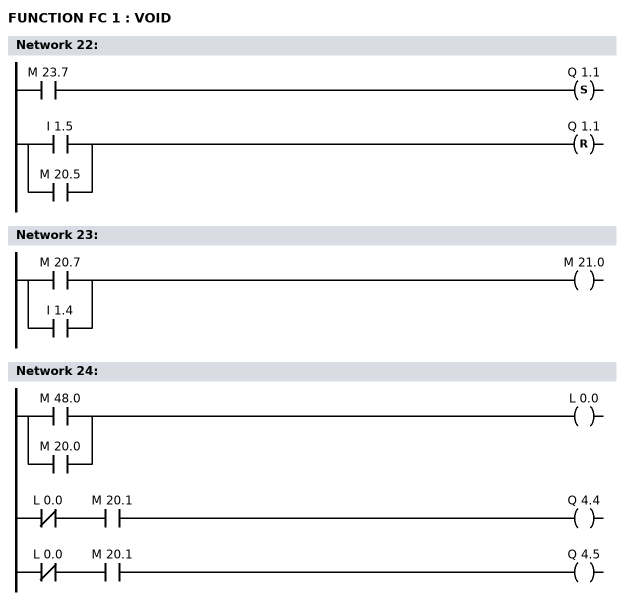

      A     M     23.7;
      S     Q      1.1;
      A(    ;
      O     I      1.5;
      O     M     20.5;
      )     ;
      R     Q      1.1;
      NOP   0;
NETWORK
TITLE =

      O     M     20.7;
      O     I      1.4;
      =     M     21.0;
NETWORK
TITLE =

      O     M     48.0;
      O     M     20.0;
      =     L      0.0;
      AN    L      0.0;
      A     M     20.1;
      =     Q      4.4;
      AN    L      0.0;
      A     M     20.1;
      =     Q      4.5;
NETWORK
TITLE =

      A(    ;
      A(    ;
      A     M     35.1;
      A     M     35.0;
      A     M     44.0;
      AN    M     38.3;
      FP    M     29.3;
      O(    ;
      A     I      1.2;
      FP    M     28.0;
      )     ;
      )     ;
      S     M     27.2;
      A(    ;
      AN    M     44.1;
      FP    M     47.0;
      O     T      3;
      O     M     20.7;
      O(    ;
      A     M     38.3;
      FP    M     38.7;
      )     ;
      O(    ;
      A     I      1.2;
      FP    M     29.4;
      A     Q      0.0;
      )     ;
      )     ;
      R     M     27.2;
      A     M     27.2;
      )     ;
      A     M     10.7;
      =     Q      0.0;
NETWORK
TITLE =

      A     M     27.2;
      L     DB2.DBW    4;
      SD    T      2;
      NOP   0;
      NOP   0;
      NOP   0;
      A     T      2;
      =     M     27.3;
NETWORK
TITLE =

      A(    ;
      A     M     27.2;
      L     DB2.DBW   10;
      SD    T      5;
      NOP   0;
      NOP   0;
      NOP   0;
      A     T      5;
      )     ;
      L     DB2.DBW    6;
      SE    T      3;
      NOP   0;
      NOP   0;
      NOP   0;
      NOP   0;
NETWORK
TITLE =

      CALL FC     3 ;
      NOP   0;
NETWORK
TITLE =

      CALL FC    10 ;
      NOP   0;
END_FUNCTION

FUNCTION FC 18 : VOID
TITLE =
AUTHOR : Xaadem <yalanci63@yahoo.com>
FAMILY : CONTROL
NAME : CONTROL
VERSION : 0.1

BEGIN
NETWORK
TITLE =

      A     Q      6.3;
      A     M     20.1;
      =     L      0.0;
      A     L      0.0;
      JNB   M001;
      L     DB4.DBD    8;
      L     -1.000000e+000;
      *R    ;
      T     DB4.DBD   16;
M001: NOP   0;
      AN    L      0.0;
      JNB   M002;
      L     DB4.DBD    8;
      L     1.000000e+000;
      *R    ;
      T     DB4.DBD   16;
M002: NOP   0;
NETWORK
TITLE =
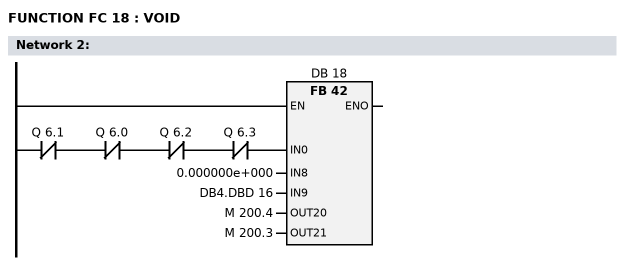

      AN    Q      6.1;
      AN    Q      6.0;
      AN    Q      6.2;
      AN    Q      6.3;
      =     L      0.0;
      BLD   103;
      CALL FB    42 , DB    18 (
           IN0                      := L      0.0,
           IN8                      := 0.000000e+000,
           IN9                      := DB4.DBD   16,
           OUT20                    := M    200.4,
           OUT21                    := M    200.3);

      NOP   0;
END_FUNCTION

FUNCTION FC 186 : VOID
TITLE =
AUTHOR : Xaadem <yalanci63@yahoo.com>
FAMILY : GENERAL
NAME : BYTECOMP
VERSION : 0.0


VAR_INPUT
  IN0 : BYTE ;
  IN1 : BYTE ;
END_VAR
VAR_OUTPUT
  OUT2 : BOOL ;
  OUT3 : BOOL ;
  OUT4 : BOOL ;
  OUT5 : BOOL ;
END_VAR
VAR_TEMP
  TEMP6 : INT ;
  TEMP7 : INT ;
END_VAR
BEGIN
NETWORK
TITLE =
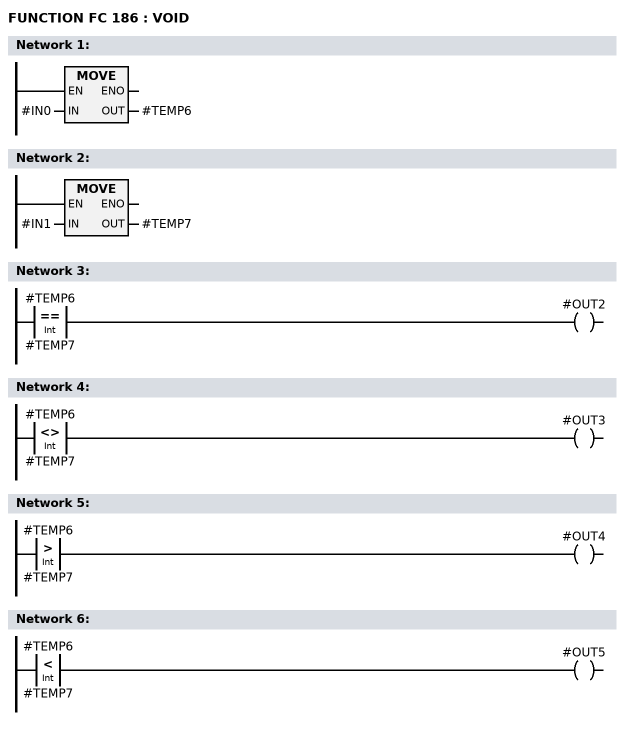

      L     #IN0;
      T     #TEMP6;
      NOP   0;
NETWORK
TITLE =

      L     #IN1;
      T     #TEMP7;
      NOP   0;
NETWORK
TITLE =

      L     #TEMP6;
      L     #TEMP7;
      ==I   ;
      =     #OUT2;
NETWORK
TITLE =

      L     #TEMP6;
      L     #TEMP7;
      <>I   ;
      =     #OUT3;
NETWORK
TITLE =

      L     #TEMP6;
      L     #TEMP7;
      >I    ;
      =     #OUT4;
NETWORK
TITLE =

      L     #TEMP6;
      L     #TEMP7;
      <I    ;
      =     #OUT5;
END_FUNCTION

ORGANIZATION_BLOCK OB 1
TITLE =
AUTHOR : Xaadem <yalanci63@yahoo.com>
VERSION : 0.1


VAR_TEMP
  TEMP0 : BYTE ;
  TEMP1 : BYTE ;
  TEMP2 : BYTE ;
  TEMP3 : BYTE ;
  TEMP4 : BYTE ;
  TEMP5 : BYTE ;
  TEMP6 : INT ;
  TEMP7 : INT ;
  TEMP8 : INT ;
  TEMP9 : DATE_AND_TIME ;
  TEMP10 : WORD ;
END_VAR
BEGIN
NETWORK
TITLE =

      CALL FC   186 (
           IN0                      := #TEMP1,
           IN1                      := B#16#1,
           OUT2                     := M     20.5,
           OUT3                     := M     20.2,
           OUT4                     := M     20.2,
           OUT5                     := M     20.2);
      NOP   0;
NETWORK
TITLE =

      CALL FC     1 ;
      NOP   0;
END_ORGANIZATION_BLOCK

ORGANIZATION_BLOCK OB 35
VERSION : 0.0


VAR_TEMP
  TEMP0 : BYTE ;
  TEMP1 : BYTE ;
  TEMP2 : BYTE ;
  TEMP3 : BYTE ;
  TEMP4 : BYTE ;
  TEMP5 : BYTE ;
  TEMP6 : WORD ;
  TEMP7 : INT ;
  TEMP8 : INT ;
  TEMP9 : DATE_AND_TIME ;
END_VAR
BEGIN
NETWORK
TITLE =

      CALL FC    18 ;
      NOP   0;
END_ORGANIZATION_BLOCK

ORGANIZATION_BLOCK OB 85
VERSION : 0.0


VAR_TEMP
  TEMP0 : BYTE ;
  TEMP1 : BYTE ;
  TEMP2 : BYTE ;
  TEMP3 : BYTE ;
  TEMP4 : BYTE ;
  TEMP5 : BYTE ;
  TEMP6 : INT ;
  TEMP7 : BYTE ;
  TEMP8 : BYTE ;
  TEMP9 : BYTE ;
  TEMP10 : BYTE ;
  TEMP11 : DATE_AND_TIME ;
END_VAR
BEGIN
END_ORGANIZATION_BLOCK

ORGANIZATION_BLOCK OB 86
VERSION : 0.0


VAR_TEMP
  TEMP0 : BYTE ;
  TEMP1 : BYTE ;
  TEMP2 : BYTE ;
  TEMP3 : BYTE ;
  TEMP4 : BYTE ;
  TEMP5 : BYTE ;
  TEMP6 : WORD ;
  TEMP7 : ARRAY  [0 .. 31 ] OF BOOL ;
  TEMP8 : DATE_AND_TIME ;
END_VAR
BEGIN
END_ORGANIZATION_BLOCK

ORGANIZATION_BLOCK OB 122
VERSION : 0.0


VAR_TEMP
  TEMP0 : BYTE ;
  TEMP1 : BYTE ;
  TEMP2 : BYTE ;
  TEMP3 : BYTE ;
  TEMP4 : BYTE ;
  TEMP5 : BYTE ;
  TEMP6 : WORD ;
  TEMP7 : WORD ;
  TEMP8 : WORD ;
  TEMP9 : DATE_AND_TIME ;
END_VAR
BEGIN
END_ORGANIZATION_BLOCK

